# EPICS autosave request: support/ebrick/2-2-3/iocBoot/iocebrick/autosave/ebrickDIOinp.req
$(P)$(H)$(F)$(D).SCAN
$(P)$(H)$(F)$(D).DESC
